(* Logix 5000 project; controller PLCNo1 vendor 1 type 14 code 196 rev 35.11; software revision 35.00 *)

TASK MainTask (continuous, watchdog 500 ms) : MainProgram

MODULES
   Local : vendor 1 type 14 code 196 (5069 0, rev 35.11)
      PLCNo2 : vendor 1 type 14 code 196 (Ethernet 192.168.1.2, rev 35.1)
      ETAP : 1783-ETAP (Ethernet 192.168.1.101, rev 2.1)
      RPLC : 5094-AENTR (Ethernet 192.168.1.11, rev 4.1)
END_MODULES

ADD_ON_INSTRUCTION Seal_In_Logic   (* revision 1.0 *)
VAR_INPUT
   Start : BOOL; {required}
   Stop : BOOL; {required}
   running : BOOL; {visible}
END_VAR
VAR
   time_to_run : TIMER; {access None}
   ONS_Start : BOOL; {access None}
END_VAR

ROUTINE Logic   (* ladder *)
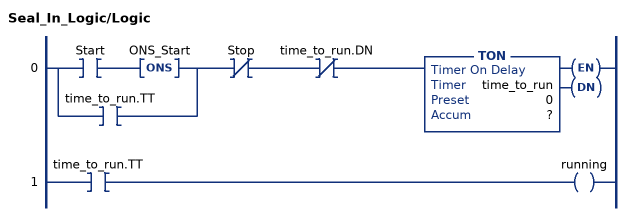
   0: [XIC(Start) ONS(ONS_Start) ,XIC(time_to_run.TT) ]XIO(Stop)XIO(time_to_run.DN)TON(time_to_run,?,?);
   1: XIC(time_to_run.TT)OTE(running);
END_ROUTINE
END_ADD_ON_INSTRUCTION

PROGRAM MainProgram   (* main routine MainRoutine *)
VAR
   control : Seal_In_Logic;
   MSG : MESSAGE;
        MessageParameters(ServiceCode := 16#000e, DestinationTag := MSG_Value, ...)
   MSG_Value : DINT;
   out : BOOL;
   start_lab_1 : BOOL;
   start_lab_2 : BOOL;
   start_lab_3 : BOOL := 1;
   stop_lab_3 : BOOL;
   TimeOfDay : date_and_time;
END_VAR

ROUTINE MainRoutine   (* ladder *)
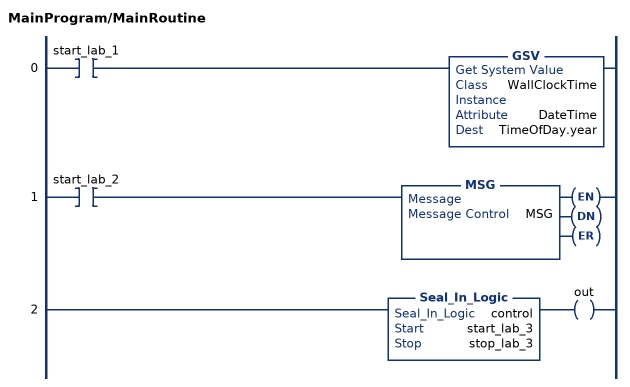
   0: XIC(start_lab_1)GSV(WallClockTime,,DateTime,TimeOfDay.year);
   1: XIC(start_lab_2)MSG(MSG);
   2: Seal_In_Logic(control,start_lab_3,stop_lab_3)OTE(out);
END_ROUTINE
END_PROGRAM
